FUNCTION MatInv3 : ARRAY [0..2,0..2] OF LREAL
VAR_INPUT
	A : ARRAY [0..2,0..2] OF LREAL;
END_VAR

VAR
	det		: LREAL;
END_VAR

det := MatDet3(A);

MatInv3[0,0] := ( A[1,1]*A[2,2] - A[1,2]*A[2,1] ) / det;
MatInv3[0,1] := ( -A[0,1]*A[2,2] + A[0,2]*A[2,1] ) / det;
MatInv3[0,2] := ( A[0,1]*A[1,2] - A[0,2]*A[1,1] ) / det;
MatInv3[1,0] := ( -A[1,0]*A[2,2] + A[1,2]*A[2,0] ) / det;
MatInv3[1,1] := ( A[0,0]*A[2,2] - A[0,2]*A[2,0] ) / det;
MatInv3[1,2] := ( -A[0,0]*A[1,2] + A[0,2]*A[1,0] ) / det;
MatInv3[2,0] := ( A[1,0]*A[2,1] - A[1,1]*A[2,0] ) / det;
MatInv3[2,1] := ( -A[0,0]*A[2,1] + A[0,1]*A[2,0] ) / det;
MatInv3[2,2] := ( A[0,0]*A[1,1] - A[0,1]*A[1,0] ) / det;

END_FUNCTION

(* stored: Version 1.1.0.1, ProductVersion 3.1.4024.11
   POU MatInv3: Id {19f7f81c-5e31-4a68-8e21-e9f3e97b1c66}, SpecialFunc None *)
